// TIA Portal V19 export
VAR_GLOBAL   // PLC tag table "Parameterwaardes"
END_VAR
VAR_GLOBAL CONSTANT   // user constants
   Ja : USInt := 11;
   Aan : USInt := 12;
   Open : USInt := 13;
   Beschikbaar : USInt := 14;
   InDienst : USInt := 16;
   Bevestiging : USInt := 17;
   OK : USInt := 18;
   Geactiveerd : USInt := 19;
   Auto : USInt := 128;
   Manueel : USInt := 129;
   Hand : USInt := 130;
   Sensorregeling : USInt := 112;
   Uit : USInt := 42;
   Bereikt : USInt := 15;
   Beperkt : USInt := 21;
   Gedeeltelijk : USInt := 22;
   InTransitie : USInt := 23;
   OpenVerlaten : USInt := 24;
   DeelsAfgesloten : USInt := 25;
   Onbepaald : USInt := 26;
   Nee : USInt := 41;
   Dicht : USInt := 43;
   NietBeschikbaar : USInt := 44;
   Storing : USInt := 45;
   OnvoorwaardelijkDicht : USInt := 46;
   Geen : USInt := 47;
   UitDienst : USInt := 48;
   Annulering : USInt := 49;
   Fout : USInt := 50;
   NietBereikt : USInt := 51;
   Onderdrukt : USInt := 52;
   Stop : USInt := 53;
   Overbrugd : USInt := 54;
   NOK : USInt := 55;
   Gedeactiveerd : USInt := 56;
   Gedoofd : USInt := 61;
   Rood : USInt := 62;
   GeelKnipper : USInt := 63;
   Geel : USInt := 64;
   Groen : USInt := 65;
   Leeg : USInt := 70;
   LLW : USInt := 71;
   LW : USInt := 72;
   SW : USInt := 73;
   MSW : USInt := 74;
   LHW : USInt := 75;
   HHW : USInt := 76;
   Rijrichting : USInt := 81;
   Hoog : USInt := 82;
   Max : USInt := 83;
   Gent : USInt := 84;
   Oplopend : USInt := 85;
   Dag : USInt := 86;
   Tegenrij : USInt := 91;
   Laag : USInt := 92;
   Min : USInt := 93;
   Luik : USInt := 94;
   Aflopend : USInt := 95;
   Nacht : USInt := 96;
   Lokaal : USInt := 101;
   Centraal : USInt := 102;
   Licht : USInt := 105;
   Matig : USInt := 106;
   Waarneembaar : USInt := 107;
   Ernstig : USInt := 108;
   Regeling : USInt := 111;
   Windmeting : USInt := 113;
   Bewaken : USInt := 115;
   Blussen : USInt := 116;
   Testen : USInt := 117;
   Klein : USInt := 120;
   Groot : USInt := 121;
   NietSel : USInt := 125;
   SelHand : USInt := 126;
   SelAuto : USInt := 127;
   Reset : USInt := 135;
   Parallel : USInt := 137;
   Eiland : USInt := 138;
   Live : USInt := 140;
   Boodschap : USInt := 141;
   Radio : USInt := 142;
   Gesprek : USInt := 145;
   Wacht : USInt := 146;
   Aanvraag : USInt := 147;
   Recirculatie : USInt := 150;
   Bergen : USInt := 153;
   LeegHouden : USInt := 154;
   Lozen : USInt := 155;
   OnderWater : USInt := 157;
   BovenWater : USInt := 158;
   Onderhoud : USInt := 160;
   Normaal : USInt := 161;
   Calamiteit : USInt := 162;
   StandBy : USInt := 163;
   Ondersteunend : USInt := 164;
   Evacuatie : USInt := 165;
   Vlucht : USInt := 166;
   Brand : USInt := 167;
   Waarschuw : USInt := 168;
   "TSCT+GL" : USInt := 200;   // Tunnelkoker van Gent naar Luik
   "TSCT+LG" : USInt := 201;   // Tunnelkoker van Luik naar Gent
   "TOKA+BR" : USInt := 202;   // Tunnelkoker van Brussel naar Rotterdam
   "TOKA+RB" : USInt := 203;   // Tunnelkoker van Rotterdam naar Brussel
   "TLUC+AR" : USInt := 204;   // Tunnelkoker van Antwerpen naar Rotterdam
   "TLUC+BA" : USInt := 205;   // Tunnelkoker van Brussel naar Antwerpen
   "TLUC+BR" : USInt := 206;   // Tunnelkoker van Brussel naar Rotterdam
   "TLUC+RA" : USInt := 207;   // Tunnelkoker van Rotterdam naar Antwerpen
   "TLUC+RB" : USInt := 208;   // Tunnelkoker van Rotterdam naar Brussel
   "TLUC+AB" : USInt := 209;   // Tunnelkoker van Antwerpen naar Brussel
   "TKZO+GR" : USInt := 210;   // Tunnelkoker van Gent naar Rotterdam
   "TKZO+RG" : USInt := 211;   // Tunnelkoker van Rotterdam naar Gent
   "TKZB+LG" : USInt := 212;   // Tunnelkoker van Luik naar Gent
   "TKZB+GL" : USInt := 213;   // Tunnelkoker van Gent naar Luik
   "TSCH+BR" : USInt := 214;   // Tunnelkoker van Brussel naar Rotterdam
   "TSCH+RB" : USInt := 215;   // Tunnelkoker van Rotterdam naar Brussel
   "TKZO+RA" : USInt := 216;   // Uitrit van Rotterdam naar Antwerpen
   "TKZO+AR" : USInt := 217;   // Inrit van Antwerpen naar Rotterdam
   "TKZB+KA" : USInt := 218;   // Uitrit kanalzone knooppunt naar Antwerpen
   "TKZB+LK" : USInt := 219;   // Uitrit luik naar kanaalzone knooppunt
   "TKZB+AK" : USInt := 220;   // Inrit antwerpen naar kanaalzone knooppunt
   "TKZB+KL" : USInt := 221;   // Inrit kanaalzone knooppunt naar Luik
END_VAR
